FUNCTION_BLOCK "FbFilterNaN"
TITLE = 'Фильтр NaN и Inf для чисел REAL.'

{ S7_read_back := 'true' ;
  S7_blockview := 'big'  }

AUTHOR  : VA
FAMILY  : LIB_PLC
VERSION : '2.2'

VAR_INPUT // Входные переменные, сохраняемые.
In       :REAL := 0.0; // Вход.
ErrValue :REAL := 0.0  ; // Значение для Out при не корректном значении на входе In.
END_VAR

VAR_OUTPUT // Выходные переменные, сохраняемые.
Out :REAL := 0.0  ; // Выход.
Err :BOOL := FALSE; // Флаг ошибки.
END_VAR

VAR // Внутренние переменные, сохраняемые.
Flag_nan_1   :BOOL := FALSE ; // Флаг не число метод 1, по стандарту IEEE 754.
Flag_nan_2   :BOOL := FALSE ; // Флаг не число метод 2, как в GCC.
Flag_nan_3   :BOOL := FALSE ; // Флаг не число метод 3, математическое определение.
Flag_pos_inf :BOOL := FALSE ; // Флаг плюс бесконечность, математическое определение.
Flag_neg_inf :BOOL := FALSE ; // Флаг минус бесконечность, математическое определение.
ZERO         :REAL := 0.0   ; // 0 CONST
END_VAR

BEGIN

// Фильтр NaN и Inf для чисел REAL.
//      DbFilterNaN
//    +-------------+
//    | FbFilterNaN |
// ->-|In        Out|->-
//   -|ErrValue  Err|-
//    +-------------+

// Если In==(NaN или Inf или -Inf) то Out=0 иначе Out=In.
// DW#16#7F800000=DW#2#01111111_10000000_00000000_00000000
// Стандарт IEEE 754.
ZERO := 0.0;
Flag_nan_1   := ((REAL_TO_DWORD(In) AND DW#16#7F800000) = DW#16#7F800000);
Flag_nan_2   := (In <> In);
Flag_nan_3   := ((ZERO / ZERO) = In);
Flag_pos_inf := (( 1.0 / ZERO) = In);
Flag_neg_inf := ((-1.0 / ZERO) = In);

Err := Flag_nan_1 OR Flag_nan_2 OR Flag_nan_3 OR Flag_pos_inf OR Flag_neg_inf;

IF (Err) THEN
Out := ErrValue;
// По умолчанию при ошибке на выходе будит 0.
// Если хотим показать последнее значение без ошибки то,
// при вызове данного блока сделать петлю с выхода на так:
// DbFilterNaN1.ErrValue := DbFilterNaN1.Out
// DbFilterNaN1();
ELSE
// Штатный режим работы без ошибок.
Out := In;
END_IF;

// @COPYLEFT ALL WRONGS RESERVED :)
// Author: VA
// Contacts: DIY.PLC.314@gmail.com
// Date start LIB_PLC: 2014
// License: GNU GPL-2.0-or-later
// https://www.gnu.org/licenses/old-licenses/gpl-2.0.html
// https://www.youtube.com/watch?v=n1F_MfLRlX0
// https://www.youtube.com/@DIY_PLC
// https://github.com/DIYPLC/LIB_PLC
// https://oshwlab.com/diy.plc.314/PLC_HW1_SW1
// https://3dtoday.ru/3d-models/mechanical-parts/body/korpus-na-din-reiku
// https://t.me/DIY_PLC
// https://drive.google.com/drive/folders/16GDX0i07rwDrl_oPzL-lQAqMiAz3ouJV?usp=sharing

END_FUNCTION_BLOCK
